# EPICS substitutions: iocBoot/iocTomoScanStream_2BMB/tomoScanStream.substitutions
file "$(TOP)/db/tomoScan.template"
{
pattern
{  P,        R,          CAMERA,   FILE_PLUGIN,    ROTATION,   SAMPLE_X,  SAMPLE_Y,      CLOSE_SHUTTER,       CLOSE_VALUE,        OPEN_SHUTTER,         OPEN_VALUE}
{2bmb:, TomoScanStream:, 2bmbSP2:, 2bmbSP2:HDF1:,  2bmb:m100,  2bmb:m63,  2bmb:m25,  2bma:A_shutter:close.VAL,    1,         2bma:A_shutter:open.VAL,        1}
}

# For the Ensemble PSO_ENC_PER_ROTATION is a signed number containing the number of encoder pulses per rotation in positive dial coordinates
file "$(TOP)/db/tomoScan_PSO.template"
{
pattern
{  P,          R,       PSO_MODEL,  PSO_PORT, PSO_AXIS_NAME, PSO_ENC_INPUT, PSO_ENC_PER_ROTATION}
{2bmb:, TomoScanStream:,    0,      PSO_PORT,      X,             3,            720000.}
}

file "$(TOP)/db/tomoScan_2BM.template"
{
pattern
{  P,          R,              BEAM_READY,      READY_VALUE,       CLOSE_FAST_SHUTTER,        CLOSE_FAST_VALUE,   OPEN_FAST_SHUTTER,          OPEN_FAST_VALUE,         SHUTTER_STATUS,               MCT_OPTICS}
{2bmb:, TomoScanStream:,   ACIS:ShutterPermit,       1,          2bma:B_shutter:close.VAL,            1,          2bma:B_shutter:open.VAL,             1,           PA:02BM:STA_A_FES_OPEN_PL,       2bm:MCTOptics:}
}

file "$(TOP)/db/tomoScanStream.template"
{
pattern
{  P,        R,           PVA_PLUGIN,     ROI_PLUGIN,     CB_PLUGIN,          PVA_STREAM,}
{2bmb:, TomoScanStream:, 2bmbSP2:Pva1:,  2bmbSP2:ROI1:,  2bmbSP2:CB1:, 2bmb:TomoScanStream:}
}
